FUNCTION FUN_LeftZeroPadding : STRING
VAR_INPUT
	input_string : INT;
END_VAR
VAR
	temp : STRING(255);
END_VAR

temp := INT_TO_STRING(input_string);

IF LEN(temp) = 1 THEN
	FUN_LeftZeroPadding:= CONCAT('0', temp);
ELSIF LEN(temp) = 2 THEN
	FUN_LeftZeroPadding:= temp;
END_IF

END_FUNCTION

(* stored: Version 1.1.0.1, ProductVersion 3.1.4024.4
   POU FUN_LeftZeroPadding: Id {fe0f8467-f021-48db-b457-53fe813ef60d}, SpecialFunc None *)
